FUNCTION_BLOCK interResourceTxLReal (* goFB_ignore *)
  (* Standard: 61499-2 *)
  (* Version 0.1, 2017-00-25, hpea485, UOA *)
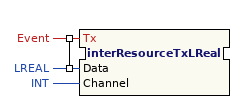
  EVENT_INPUT
    Tx WITH Data;
  END_EVENT
  VAR_INPUT
    Data : LREAL;
    Channel : INT;
  END_VAR
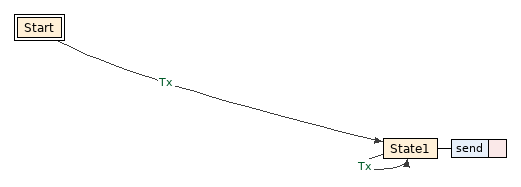
  EC_STATES
    Start;
    State1 : send;
  END_STATES
  EC_TRANSITIONS
    Start TO State1 := Tx;
    State1 TO State1 := Tx;
  END_TRANSITIONS
  ALGORITHM send IN C:
something;
something;
  END_ALGORITHM
END_FUNCTION_BLOCK
